// TIA Portal V20 export
// export: Created 2025-12-01T14:56:48.2327628Z, ExportSetting None, DisplayName Totally Integrated Automation Portal, DisplayVersion V20 Update 3, DisplayName TIA Portal Openness, DisplayVersion V20 Update 3, DisplayName TIA Portal Version Control Interface, DisplayVersion V20 Update 3, DisplayName STEP 7 Professional, DisplayVersion V20 Update 3, DisplayName STEP 7 Safety, DisplayVersion V20 Update 2, DisplayName WinCC Basic/Comfort/Advanced, DisplayVersion V20 Update 3, DisplayName WinCC Professional, DisplayVersion V20 Update 3, DisplayName WinCC Unified, DisplayVersion V20 Update 3
FUNCTION_BLOCK "FB364_Mesa_ApiladorBandejas_ULMA"   // FB364, LAD
TITLE = Control del Ramal de Salidas
{ S7_Optimized_Access := 'FALSE' }
AUTHOR : TE_FSS
NAME : 20160211
VERSION : 3.2
// stored: AutoNumber false, SetENOAutomatically false
   VAR_INPUT
      Mesa : UInt;   // Mesa de la FB
      Error_Tx : Bool;   // Error en el Tx
      pHsMx : Bool;   // pHs de la Mesa
      Avance_Tx : Bool;   // Avance de Tx
      TP_Up : Bool;   // Detector de TP Arriba
      TP_Down : Bool;   // Detector de TP Abajo
      PRV_AVTF_Bandeja : Bool;   // E1 >> Aviso de Entrada de Bandeja
      PRV_AVTF_Pila_Bandejas : Bool;   // E1 >> Aviso de Entrada de Pila
      NXT_Carga_OK : Bool;   // S3 >> Permiso de Salida
      DejarCargaEnMesa : Bool;   // Dejar la Bandeja En la Mesa
      V_pHsMx : Int;   // Valor de Presencia
      V_ApHsMx : Int;   // Valor de Ausencia
      V_TOut_Atasco : Int;   // Valor de TimeOut de Entrada
      V_TOut_TP : Int;   // Valor de TmeOut de Tope
      V_Vaciado : Int;   // Valor de Vaciado
   END_VAR
   VAR_OUTPUT
      PRV_Carga_OK : Bool;   // E1 >> Permiso de Entrada
      NXT_AVTF_Bandeja : Bool;   // S3 >> Aviso de Salida de Bandeja
      NXT_AVTF_Pila : Bool;   // S3 >> Aviso de Salida de Pila
   END_VAR
   VAR_IN_OUT
      Ord_ApilarBandeja : Bool;   // Orden de Apilar Bandeja
      Ord_SalidaPila : Bool;   // Orden de Salida de Pila
   END_VAR
   VAR
      Mx_ET00 : Bool;
      Mx_ET01 : Bool;
      Mx_ET02 : Bool;
      Mx_ET10 : Bool;
      Mx_ET11 : Bool;
      Mx_ET50 : Bool;   // Descarga de Bandeja
      Mx_ET51 : Bool;   // Descarga de Bandeja
      Mx_ET60 : Bool;   // Ciclo Apilado
      Mx_ET61 : Bool;   // Ciclo Apilado
      Mx_ET70 : Bool;   // Descarga De Pila de Bandejas
      Mx_ET71 : Bool;   // Descarga De Pila de Bandejas
      STAT_NXT_AVTF_Bandeja : Bool;   // Interna >> Aviso de Salida de Bandeja
      STAT_NXT_AVTF_Pila : Bool;   // Interna >> Aviso de Salida de Pila
      MA_Avanzar_Tx : Bool;
      MA_Parar_Tx : Bool;
      MA_Subir_TP : Bool;
      MA_Bajar_TP : Bool;
      CNT_pHsMx { S7_SetPoint := 'True'} : "FB910_CNT_UHS";
      CNT_ApHsMx { S7_SetPoint := 'True'} : "FB910_CNT_UHS";
      TMP_Vaciado { S7_SetPoint := 'True'} : "FB910_CNT_UHS";
      TOut_Atasco { S7_SetPoint := 'True'} : "FB910_CNT_UHS";
      TOut_Subir_TP { S7_SetPoint := 'True'} : "FB910_CNT_UHS";
      TOut_Bajar_TP { S7_SetPoint := 'True'} : "FB910_CNT_UHS";
   END_VAR
   VAR_TEMP
      EstadoZona : "EstadoZona";   // Estado de Zona de la Mesa
      EstadoVI : "EstadosMesa";   // Estado del Vehiculo Inteliguente de la Mesa
      ConfigFB : "UDT_ConfigFB";   // Configuracion de la FB de la Mesa
      Aux_ET00 : Bool;
   END_VAR
BEGIN

REGION Network 1: INICIALIZAR - Recoger las Variables de Estado de la Mesa
   // Se recoge - Estado_CBx
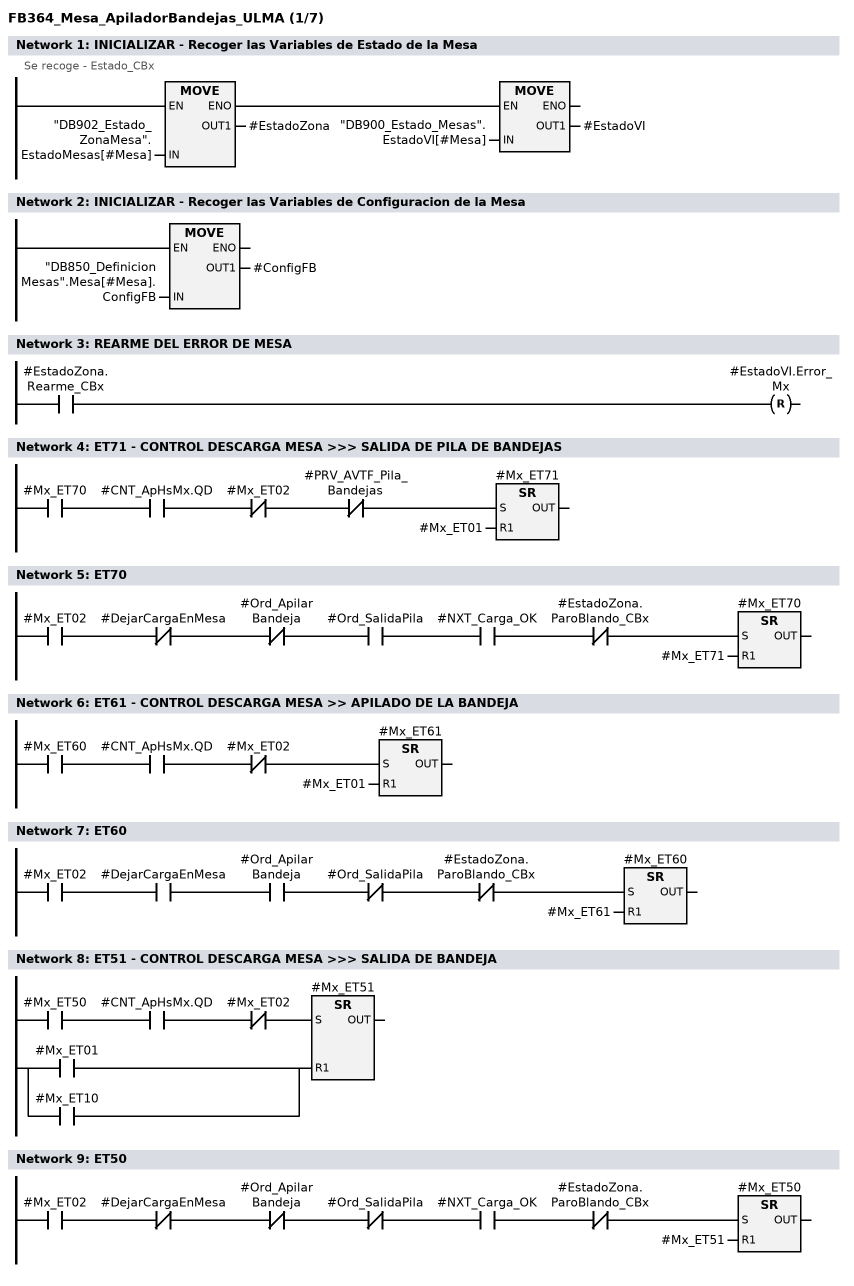
   RUNG wire#powerrail
      Move(in := "DB902_Estado_ZonaMesa".EstadoMesas[#Mesa], out1 => #EstadoZona)
      Move(in := "DB900_Estado_Mesas".EstadoVI[#Mesa], out1 => #EstadoVI)
   END_RUNG
   // the same network as SCL:
   #EstadoZona := "DB902_Estado_ZonaMesa".EstadoMesas[#Mesa];
   #EstadoVI := "DB900_Estado_Mesas".EstadoVI[#Mesa];
END_REGION

REGION Network 2: INICIALIZAR - Recoger las Variables de Configuracion de la Mesa
   RUNG wire#powerrail
      Move(in := "DB850_DefinicionMesas".Mesa[#Mesa].ConfigFB, out1 => #ConfigFB)
   END_RUNG
   // the same network as SCL:
   #ConfigFB := "DB850_DefinicionMesas".Mesa[#Mesa].ConfigFB;
END_REGION

REGION Network 3: REARME DEL ERROR DE MESA
   RUNG wire#powerrail
      Contact( #EstadoZona.Rearme_CBx )
      R_Coil( #EstadoVI.Error_Mx )
   END_RUNG
   // the same network as SCL:
   IF #EstadoZona.Rearme_CBx THEN #EstadoVI.Error_Mx := FALSE; END_IF;
END_REGION

REGION Network 4: ET71 - CONTROL DESCARGA MESA >>> SALIDA DE PILA DE BANDEJAS
   RUNG wire#powerrail
      Contact( #Mx_ET70 )
      Contact( #CNT_ApHsMx.QD )
      I_Contact( #Mx_ET02 )
      I_Contact( #PRV_AVTF_Pila_Bandejas )
      S_SR(operand := #Mx_ET71, r1 := #Mx_ET01)
   END_RUNG
   // the same network as SCL:
   IF #Mx_ET70 AND #CNT_ApHsMx.QD AND NOT #Mx_ET02 AND NOT #PRV_AVTF_Pila_Bandejas THEN
       #Mx_ET71 := TRUE;   // SR flip-flop
   END_IF;
   IF #Mx_ET01 THEN #Mx_ET71 := FALSE; END_IF;
END_REGION

REGION Network 5: ET70
   RUNG wire#powerrail
      Contact( #Mx_ET02 )
      I_Contact( #DejarCargaEnMesa )
      I_Contact( #Ord_ApilarBandeja )
      Contact( #Ord_SalidaPila )
      Contact( #NXT_Carga_OK )
      I_Contact( #EstadoZona.ParoBlando_CBx )
      S_SR(operand := #Mx_ET70, r1 := #Mx_ET71)
   END_RUNG
   // the same network as SCL:
   IF #Mx_ET02 AND NOT #DejarCargaEnMesa AND NOT #Ord_ApilarBandeja AND #Ord_SalidaPila AND #NXT_Carga_OK AND NOT #EstadoZona.ParoBlando_CBx THEN
       #Mx_ET70 := TRUE;   // SR flip-flop
   END_IF;
   IF #Mx_ET71 THEN #Mx_ET70 := FALSE; END_IF;
END_REGION

REGION Network 6: ET61 - CONTROL DESCARGA MESA >> APILADO DE LA BANDEJA
   RUNG wire#powerrail
      Contact( #Mx_ET60 )
      Contact( #CNT_ApHsMx.QD )
      I_Contact( #Mx_ET02 )
      S_SR(operand := #Mx_ET61, r1 := #Mx_ET01)
   END_RUNG
   // the same network as SCL:
   IF #Mx_ET60 AND #CNT_ApHsMx.QD AND NOT #Mx_ET02 THEN
       #Mx_ET61 := TRUE;   // SR flip-flop
   END_IF;
   IF #Mx_ET01 THEN #Mx_ET61 := FALSE; END_IF;
END_REGION

REGION Network 7: ET60
   RUNG wire#powerrail
      Contact( #Mx_ET02 )
      Contact( #DejarCargaEnMesa )
      Contact( #Ord_ApilarBandeja )
      I_Contact( #Ord_SalidaPila )
      I_Contact( #EstadoZona.ParoBlando_CBx )
      S_SR(operand := #Mx_ET60, r1 := #Mx_ET61)
   END_RUNG
   // the same network as SCL:
   IF #Mx_ET02 AND #DejarCargaEnMesa AND #Ord_ApilarBandeja AND NOT #Ord_SalidaPila AND NOT #EstadoZona.ParoBlando_CBx THEN
       #Mx_ET60 := TRUE;   // SR flip-flop
   END_IF;
   IF #Mx_ET61 THEN #Mx_ET60 := FALSE; END_IF;
END_REGION

REGION Network 8: ET51 - CONTROL DESCARGA MESA >>> SALIDA DE BANDEJA
   RUNG wire#powerrail
      Contact( #Mx_ET50 )
      Contact( #CNT_ApHsMx.QD )
      I_Contact( #Mx_ET02 )
      S_SR(operand := #Mx_ET51, r1 := wire#w1)
   END_RUNG
   RUNG wire#powerrail
      Contact( #Mx_ET01 )
   END_RUNG wire#w1
   RUNG wire#powerrail
      Contact( #Mx_ET10 )
   END_RUNG wire#w1
   // the same network as SCL:
   IF #Mx_ET50 AND #CNT_ApHsMx.QD AND NOT #Mx_ET02 THEN
       #Mx_ET51 := TRUE;   // SR flip-flop
   END_IF;
   IF #Mx_ET01 OR #Mx_ET10 THEN #Mx_ET51 := FALSE; END_IF;
END_REGION

REGION Network 9: ET50
   RUNG wire#powerrail
      Contact( #Mx_ET02 )
      I_Contact( #DejarCargaEnMesa )
      I_Contact( #Ord_ApilarBandeja )
      I_Contact( #Ord_SalidaPila )
      Contact( #NXT_Carga_OK )
      I_Contact( #EstadoZona.ParoBlando_CBx )
      S_SR(operand := #Mx_ET50, r1 := #Mx_ET51)
   END_RUNG
   // the same network as SCL:
   IF #Mx_ET02 AND NOT #DejarCargaEnMesa AND NOT #Ord_ApilarBandeja AND NOT #Ord_SalidaPila AND #NXT_Carga_OK AND NOT #EstadoZona.ParoBlando_CBx THEN
       #Mx_ET50 := TRUE;   // SR flip-flop
   END_IF;
   IF #Mx_ET51 THEN #Mx_ET50 := FALSE; END_IF;
END_REGION

REGION Network 10: ET02 - ESTADO REPOSO CARGADA
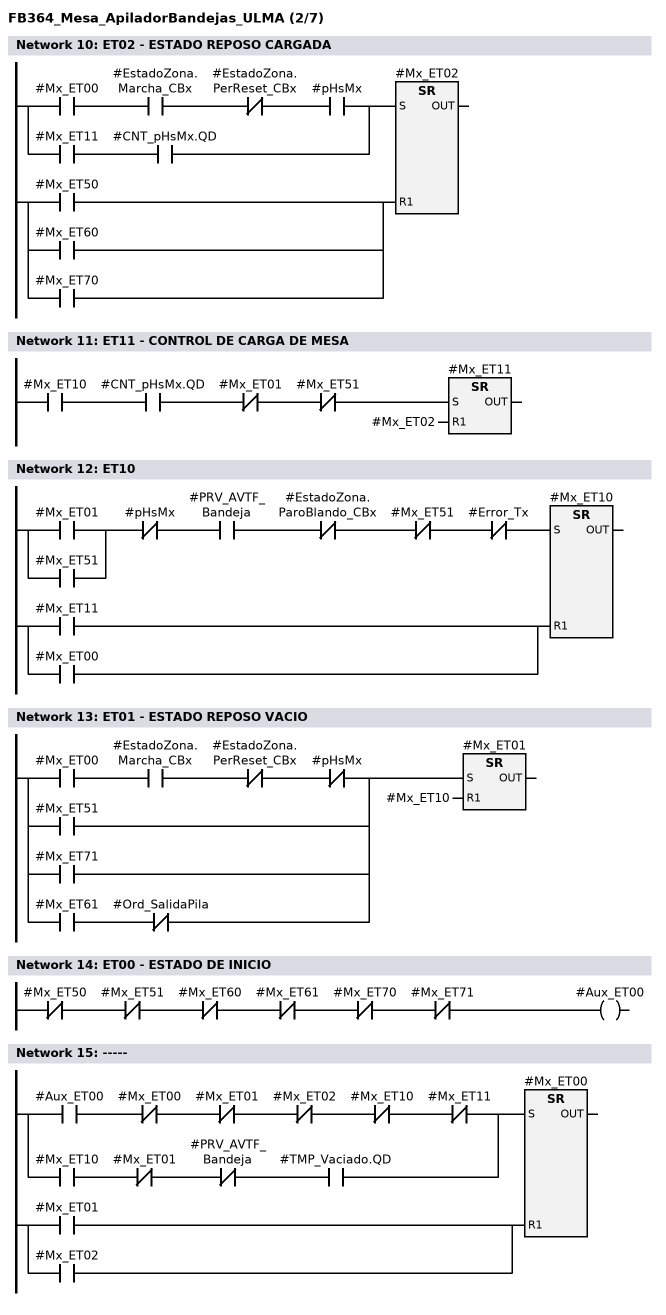
   RUNG wire#powerrail
      Contact( #Mx_ET00 )
      Contact( #EstadoZona.Marcha_CBx )
      I_Contact( #EstadoZona.PerReset_CBx )
      Contact( #pHsMx )
      wire#w1
      S_SR(operand := #Mx_ET02, r1 := wire#w2)
   END_RUNG
   RUNG wire#powerrail
      Contact( #Mx_ET11 )
      Contact( #CNT_pHsMx.QD )
   END_RUNG wire#w1
   RUNG wire#powerrail
      Contact( #Mx_ET50 )
   END_RUNG wire#w2
   RUNG wire#powerrail
      Contact( #Mx_ET60 )
   END_RUNG wire#w2
   RUNG wire#powerrail
      Contact( #Mx_ET70 )
   END_RUNG wire#w2
   // the same network as SCL:
   IF (#Mx_ET00 AND #EstadoZona.Marcha_CBx AND NOT #EstadoZona.PerReset_CBx AND #pHsMx) OR (#Mx_ET11 AND #CNT_pHsMx.QD) THEN
       #Mx_ET02 := TRUE;   // SR flip-flop
   END_IF;
   IF #Mx_ET50 OR #Mx_ET60 OR #Mx_ET70 THEN #Mx_ET02 := FALSE; END_IF;
END_REGION

REGION Network 11: ET11 - CONTROL DE CARGA DE MESA
   RUNG wire#powerrail
      Contact( #Mx_ET10 )
      Contact( #CNT_pHsMx.QD )
      I_Contact( #Mx_ET01 )
      I_Contact( #Mx_ET51 )
      S_SR(operand := #Mx_ET11, r1 := #Mx_ET02)
   END_RUNG
   // the same network as SCL:
   IF #Mx_ET10 AND #CNT_pHsMx.QD AND NOT #Mx_ET01 AND NOT #Mx_ET51 THEN
       #Mx_ET11 := TRUE;   // SR flip-flop
   END_IF;
   IF #Mx_ET02 THEN #Mx_ET11 := FALSE; END_IF;
END_REGION

REGION Network 12: ET10
   RUNG wire#powerrail
      Contact( #Mx_ET01 )
      wire#w1
      I_Contact( #pHsMx )
      Contact( #PRV_AVTF_Bandeja )
      I_Contact( #EstadoZona.ParoBlando_CBx )
      I_Contact( #Mx_ET51 )
      I_Contact( #Error_Tx )
      S_SR(operand := #Mx_ET10, r1 := wire#w2)
   END_RUNG
   RUNG wire#powerrail
      Contact( #Mx_ET51 )
   END_RUNG wire#w1
   RUNG wire#powerrail
      Contact( #Mx_ET11 )
   END_RUNG wire#w2
   RUNG wire#powerrail
      Contact( #Mx_ET00 )
   END_RUNG wire#w2
   // the same network as SCL:
   IF (#Mx_ET01 OR #Mx_ET51) AND NOT #pHsMx AND #PRV_AVTF_Bandeja AND NOT #EstadoZona.ParoBlando_CBx AND NOT #Mx_ET51 AND NOT #Error_Tx THEN
       #Mx_ET10 := TRUE;   // SR flip-flop
   END_IF;
   IF #Mx_ET11 OR #Mx_ET00 THEN #Mx_ET10 := FALSE; END_IF;
END_REGION

REGION Network 13: ET01 - ESTADO REPOSO VACIO
   RUNG wire#powerrail
      Contact( #Mx_ET00 )
      Contact( #EstadoZona.Marcha_CBx )
      I_Contact( #EstadoZona.PerReset_CBx )
      I_Contact( #pHsMx )
      wire#w1
      S_SR(operand := #Mx_ET01, r1 := #Mx_ET10)
   END_RUNG
   RUNG wire#powerrail
      Contact( #Mx_ET51 )
   END_RUNG wire#w1
   RUNG wire#powerrail
      Contact( #Mx_ET71 )
   END_RUNG wire#w1
   RUNG wire#powerrail
      Contact( #Mx_ET61 )
      I_Contact( #Ord_SalidaPila )
   END_RUNG wire#w1
   // the same network as SCL:
   IF (#Mx_ET00 AND #EstadoZona.Marcha_CBx AND NOT #EstadoZona.PerReset_CBx AND NOT #pHsMx) OR #Mx_ET51 OR #Mx_ET71 OR (#Mx_ET61 AND NOT #Ord_SalidaPila) THEN
       #Mx_ET01 := TRUE;   // SR flip-flop
   END_IF;
   IF #Mx_ET10 THEN #Mx_ET01 := FALSE; END_IF;
END_REGION

REGION Network 14: ET00 - ESTADO DE INICIO
   RUNG wire#powerrail
      I_Contact( #Mx_ET50 )
      I_Contact( #Mx_ET51 )
      I_Contact( #Mx_ET60 )
      I_Contact( #Mx_ET61 )
      I_Contact( #Mx_ET70 )
      I_Contact( #Mx_ET71 )
      Coil( #Aux_ET00 )
   END_RUNG
   // the same network as SCL:
   #Aux_ET00 := NOT #Mx_ET50 AND NOT #Mx_ET51 AND NOT #Mx_ET60 AND NOT #Mx_ET61 AND NOT #Mx_ET70 AND NOT #Mx_ET71;
END_REGION

REGION Network 15: -----
   RUNG wire#powerrail
      Contact( #Aux_ET00 )
      I_Contact( #Mx_ET00 )
      I_Contact( #Mx_ET01 )
      I_Contact( #Mx_ET02 )
      I_Contact( #Mx_ET10 )
      I_Contact( #Mx_ET11 )
      wire#w1
      S_SR(operand := #Mx_ET00, r1 := wire#w2)
   END_RUNG
   RUNG wire#powerrail
      Contact( #Mx_ET10 )
      I_Contact( #Mx_ET01 )
      I_Contact( #PRV_AVTF_Bandeja )
      Contact( #TMP_Vaciado.QD )
   END_RUNG wire#w1
   RUNG wire#powerrail
      Contact( #Mx_ET01 )
   END_RUNG wire#w2
   RUNG wire#powerrail
      Contact( #Mx_ET02 )
   END_RUNG wire#w2
   // the same network as SCL:
   IF (#Aux_ET00 AND NOT #Mx_ET00 AND NOT #Mx_ET01 AND NOT #Mx_ET02 AND NOT #Mx_ET10 AND NOT #Mx_ET11) OR (#Mx_ET10 AND NOT #Mx_ET01 AND NOT #PRV_AVTF_Bandeja AND #TMP_Vaciado.QD) THEN
       #Mx_ET00 := TRUE;   // SR flip-flop
   END_IF;
   IF #Mx_ET01 OR #Mx_ET02 THEN #Mx_ET00 := FALSE; END_IF;
END_REGION

REGION Network 16: CONTADOR DE PRESENCIA
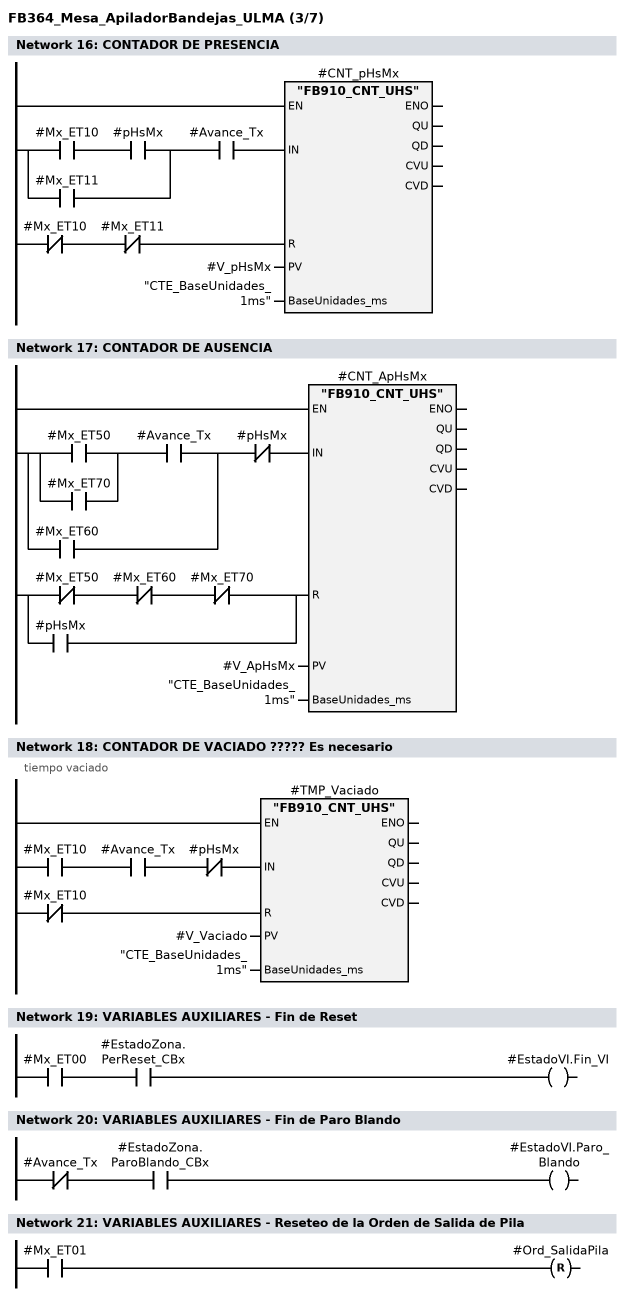
   RUNG wire#powerrail
      #CNT_pHsMx(IN := wire#w2, R := wire#w3, PV := #V_pHsMx, BaseUnidades_ms := "CTE_BaseUnidades_1ms", QU =>, QD =>, CVU =>, CVD =>)
   END_RUNG
   RUNG wire#powerrail
      Contact( #Mx_ET10 )
      Contact( #pHsMx )
      wire#w1
      Contact( #Avance_Tx )
   END_RUNG wire#w2
   RUNG wire#powerrail
      Contact( #Mx_ET11 )
   END_RUNG wire#w1
   RUNG wire#powerrail
      I_Contact( #Mx_ET10 )
      I_Contact( #Mx_ET11 )
   END_RUNG wire#w3
   // the same network as SCL:
   #CNT_pHsMx(IN := ((#Mx_ET10 AND #pHsMx) OR #Mx_ET11) AND #Avance_Tx,   // "FB910_CNT_UHS"
              R := NOT #Mx_ET10 AND NOT #Mx_ET11,
              PV := #V_pHsMx,
              BaseUnidades_ms := "CTE_BaseUnidades_1ms");
END_REGION

REGION Network 17: CONTADOR DE AUSENCIA
   RUNG wire#powerrail
      #CNT_ApHsMx(IN := wire#w3, R := wire#w4, PV := #V_ApHsMx, BaseUnidades_ms := "CTE_BaseUnidades_1ms", QU =>, QD =>, CVU =>, CVD =>)
   END_RUNG
   RUNG wire#powerrail
      Contact( #Mx_ET50 )
      wire#w1
      Contact( #Avance_Tx )
      wire#w2
      I_Contact( #pHsMx )
   END_RUNG wire#w3
   RUNG wire#powerrail
      Contact( #Mx_ET70 )
   END_RUNG wire#w1
   RUNG wire#powerrail
      Contact( #Mx_ET60 )
   END_RUNG wire#w2
   RUNG wire#powerrail
      I_Contact( #Mx_ET50 )
      I_Contact( #Mx_ET60 )
      I_Contact( #Mx_ET70 )
   END_RUNG wire#w4
   RUNG wire#powerrail
      Contact( #pHsMx )
   END_RUNG wire#w4
   // the same network as SCL:
   #CNT_ApHsMx(IN := (((#Mx_ET50 OR #Mx_ET70) AND #Avance_Tx) OR #Mx_ET60) AND NOT #pHsMx,   // "FB910_CNT_UHS"
               R := (NOT #Mx_ET50 AND NOT #Mx_ET60 AND NOT #Mx_ET70) OR #pHsMx,
               PV := #V_ApHsMx,
               BaseUnidades_ms := "CTE_BaseUnidades_1ms");
END_REGION

REGION Network 18: CONTADOR DE VACIADO ????? Es necesario
   // tiempo vaciado
   RUNG wire#powerrail
      #TMP_Vaciado(IN := wire#w1, R := wire#w2, PV := #V_Vaciado, BaseUnidades_ms := "CTE_BaseUnidades_1ms", QU =>, QD =>, CVU =>, CVD =>)
   END_RUNG
   RUNG wire#powerrail
      Contact( #Mx_ET10 )
      Contact( #Avance_Tx )
      I_Contact( #pHsMx )
   END_RUNG wire#w1
   RUNG wire#powerrail
      I_Contact( #Mx_ET10 )
   END_RUNG wire#w2
   // the same network as SCL:
   #TMP_Vaciado(IN := #Mx_ET10 AND #Avance_Tx AND NOT #pHsMx,   // "FB910_CNT_UHS"
                R := NOT #Mx_ET10,
                PV := #V_Vaciado,
                BaseUnidades_ms := "CTE_BaseUnidades_1ms");
END_REGION

REGION Network 19: VARIABLES AUXILIARES - Fin de Reset
   RUNG wire#powerrail
      Contact( #Mx_ET00 )
      Contact( #EstadoZona.PerReset_CBx )
      Coil( #EstadoVI.Fin_VI )
   END_RUNG
   // the same network as SCL:
   #EstadoVI.Fin_VI := #Mx_ET00 AND #EstadoZona.PerReset_CBx;
END_REGION

REGION Network 20: VARIABLES AUXILIARES - Fin de Paro Blando
   RUNG wire#powerrail
      I_Contact( #Avance_Tx )
      Contact( #EstadoZona.ParoBlando_CBx )
      Coil( #EstadoVI.Paro_Blando )
   END_RUNG
   // the same network as SCL:
   #EstadoVI.Paro_Blando := NOT #Avance_Tx AND #EstadoZona.ParoBlando_CBx;
END_REGION

REGION Network 21: VARIABLES AUXILIARES - Reseteo de la Orden de Salida de Pila
   RUNG wire#powerrail
      Contact( #Mx_ET01 )
      R_Coil( #Ord_SalidaPila )
   END_RUNG
   // the same network as SCL:
   IF #Mx_ET01 THEN #Ord_SalidaPila := FALSE; END_IF;
END_REGION

REGION Network 22: VARIABLES AUXILIARES - Permiso de Entrada - PRV_Carga_OK
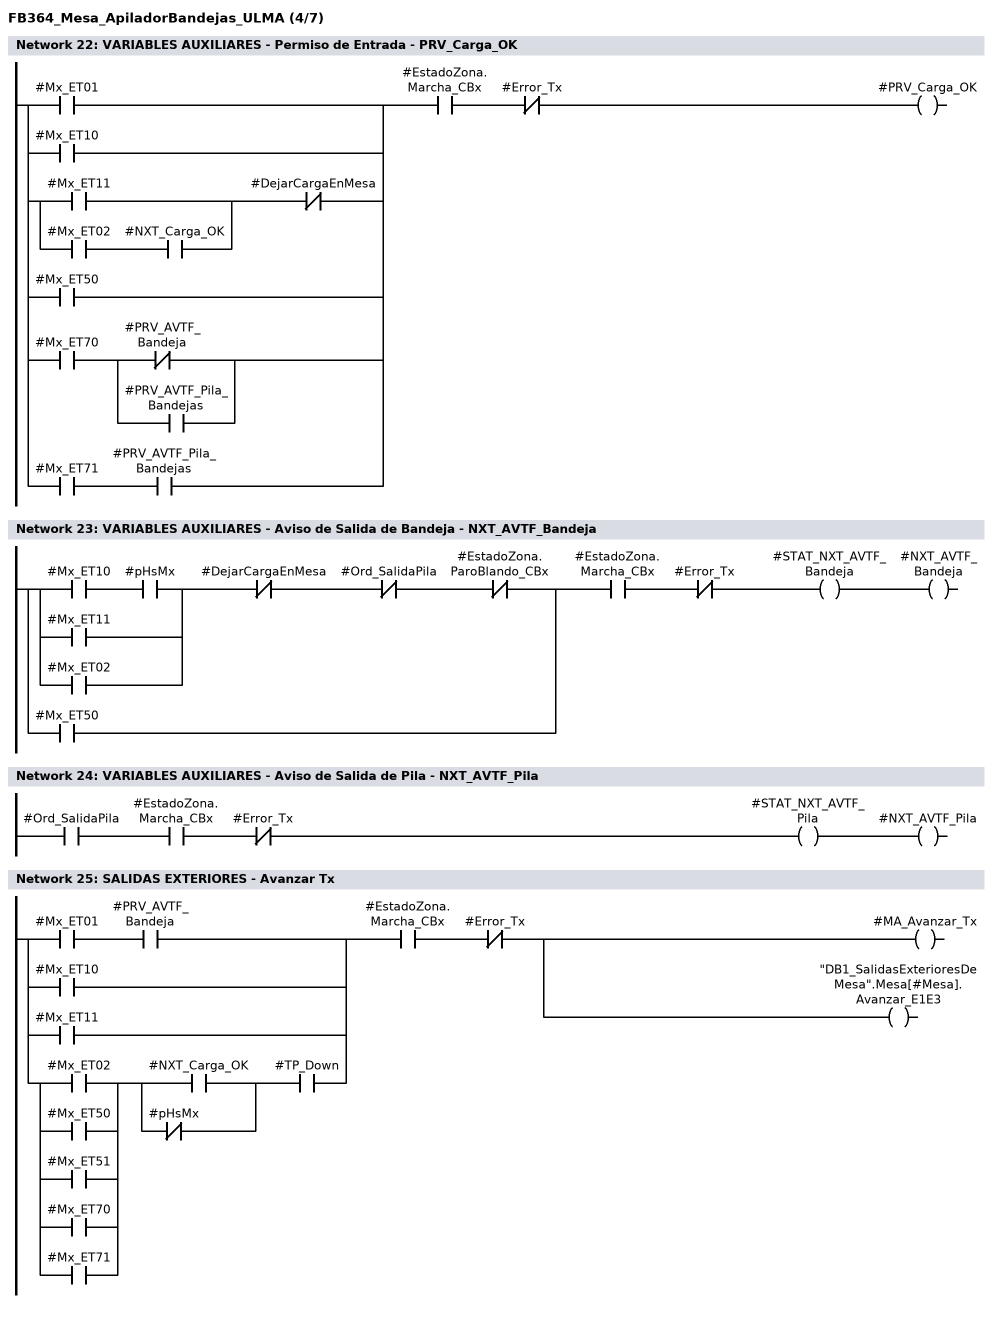
   RUNG wire#powerrail
      Contact( #Mx_ET01 )
      wire#w1
      Contact( #EstadoZona.Marcha_CBx )
      I_Contact( #Error_Tx )
      Coil( #PRV_Carga_OK )
   END_RUNG
   RUNG wire#powerrail
      Contact( #Mx_ET10 )
   END_RUNG wire#w1
   RUNG wire#powerrail
      Contact( #Mx_ET11 )
      wire#w2
      I_Contact( #DejarCargaEnMesa )
   END_RUNG wire#w1
   RUNG wire#powerrail
      Contact( #Mx_ET02 )
      Contact( #NXT_Carga_OK )
   END_RUNG wire#w2
   RUNG wire#powerrail
      Contact( #Mx_ET50 )
   END_RUNG wire#w1
   RUNG wire#powerrail
      Contact( #Mx_ET70 )
      wire#w3
      I_Contact( #PRV_AVTF_Bandeja )
   END_RUNG wire#w1
   RUNG wire#w3
      Contact( #PRV_AVTF_Pila_Bandejas )
   END_RUNG wire#w1
   RUNG wire#powerrail
      Contact( #Mx_ET71 )
      Contact( #PRV_AVTF_Pila_Bandejas )
   END_RUNG wire#w1
   // the same network as SCL:
   #PRV_Carga_OK := (#Mx_ET01 OR #Mx_ET10 OR ((#Mx_ET11 OR (#Mx_ET02 AND #NXT_Carga_OK)) AND NOT #DejarCargaEnMesa) OR #Mx_ET50 OR (#Mx_ET70 AND (NOT #PRV_AVTF_Bandeja OR #PRV_AVTF_Pila_Bandejas)) OR (#Mx_ET71 AND #PRV_AVTF_Pila_Bandejas)) AND #EstadoZona.Marcha_CBx AND NOT #Error_Tx;
END_REGION

REGION Network 23: VARIABLES AUXILIARES - Aviso de Salida de Bandeja - NXT_AVTF_Bandeja
   RUNG wire#powerrail
      Contact( #Mx_ET10 )
      Contact( #pHsMx )
      wire#w1
      I_Contact( #DejarCargaEnMesa )
      I_Contact( #Ord_SalidaPila )
      I_Contact( #EstadoZona.ParoBlando_CBx )
      wire#w2
      Contact( #EstadoZona.Marcha_CBx )
      I_Contact( #Error_Tx )
      Coil( #STAT_NXT_AVTF_Bandeja )
      Coil( #NXT_AVTF_Bandeja )
   END_RUNG
   RUNG wire#powerrail
      Contact( #Mx_ET11 )
   END_RUNG wire#w1
   RUNG wire#powerrail
      Contact( #Mx_ET02 )
   END_RUNG wire#w1
   RUNG wire#powerrail
      Contact( #Mx_ET50 )
   END_RUNG wire#w2
   // the same network as SCL:
   #STAT_NXT_AVTF_Bandeja := ((((#Mx_ET10 AND #pHsMx) OR #Mx_ET11 OR #Mx_ET02) AND NOT #DejarCargaEnMesa AND NOT #Ord_SalidaPila AND NOT #EstadoZona.ParoBlando_CBx) OR #Mx_ET50) AND #EstadoZona.Marcha_CBx AND NOT #Error_Tx;
   #NXT_AVTF_Bandeja := #STAT_NXT_AVTF_Bandeja;
END_REGION

REGION Network 24: VARIABLES AUXILIARES - Aviso de Salida de Pila - NXT_AVTF_Pila
   RUNG wire#powerrail
      Contact( #Ord_SalidaPila )
      Contact( #EstadoZona.Marcha_CBx )
      I_Contact( #Error_Tx )
      Coil( #STAT_NXT_AVTF_Pila )
      Coil( #NXT_AVTF_Pila )
   END_RUNG
   // the same network as SCL:
   #STAT_NXT_AVTF_Pila := #Ord_SalidaPila AND #EstadoZona.Marcha_CBx AND NOT #Error_Tx;
   #NXT_AVTF_Pila := #STAT_NXT_AVTF_Pila;
END_REGION

REGION Network 25: SALIDAS EXTERIORES - Avanzar Tx
   RUNG wire#powerrail
      Contact( #Mx_ET01 )
      Contact( #PRV_AVTF_Bandeja )
      wire#w1
      Contact( #EstadoZona.Marcha_CBx )
      I_Contact( #Error_Tx )
      wire#w4
      Coil( #MA_Avanzar_Tx )
   END_RUNG
   RUNG wire#powerrail
      Contact( #Mx_ET10 )
   END_RUNG wire#w1
   RUNG wire#powerrail
      Contact( #Mx_ET11 )
   END_RUNG wire#w1
   RUNG wire#powerrail
      Contact( #Mx_ET02 )
      wire#w2
      Contact( #NXT_Carga_OK )
      wire#w3
      Contact( #TP_Down )
   END_RUNG wire#w1
   RUNG wire#powerrail
      Contact( #Mx_ET50 )
   END_RUNG wire#w2
   RUNG wire#powerrail
      Contact( #Mx_ET51 )
   END_RUNG wire#w2
   RUNG wire#powerrail
      Contact( #Mx_ET70 )
   END_RUNG wire#w2
   RUNG wire#powerrail
      Contact( #Mx_ET71 )
   END_RUNG wire#w2
   RUNG wire#w2
      I_Contact( #pHsMx )
   END_RUNG wire#w3
   RUNG wire#w4
      Coil( "DB1_SalidasExterioresDeMesa".Mesa[#Mesa].Avanzar_E1E3 )
   END_RUNG
   // the same network as SCL:
   #MA_Avanzar_Tx := ((#Mx_ET01 AND #PRV_AVTF_Bandeja) OR #Mx_ET10 OR #Mx_ET11 OR ((#Mx_ET02 OR #Mx_ET50 OR #Mx_ET51 OR #Mx_ET70 OR #Mx_ET71) AND (#NXT_Carga_OK OR NOT #pHsMx) AND #TP_Down)) AND #EstadoZona.Marcha_CBx AND NOT #Error_Tx;
   "DB1_SalidasExterioresDeMesa".Mesa[#Mesa].Avanzar_E1E3 := #MA_Avanzar_Tx;
END_REGION

REGION Network 26: SALIDAS EXTERIORES - Parar Tx
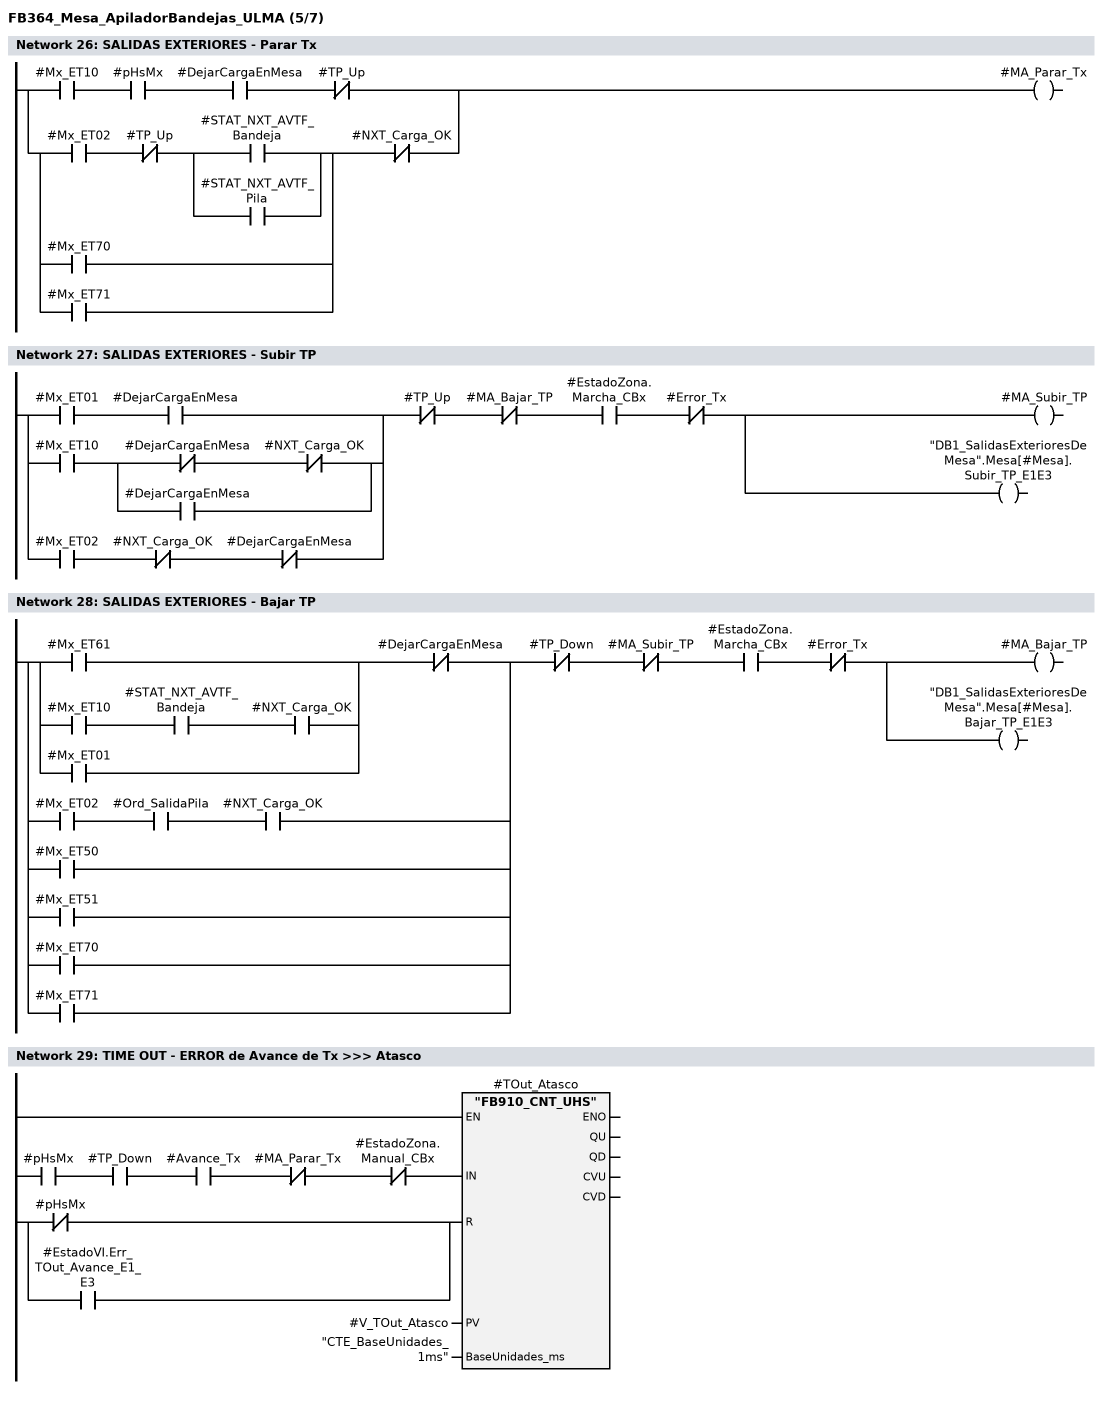
   RUNG wire#powerrail
      Contact( #Mx_ET10 )
      Contact( #pHsMx )
      Contact( #DejarCargaEnMesa )
      I_Contact( #TP_Up )
      wire#w1
      Coil( #MA_Parar_Tx )
   END_RUNG
   RUNG wire#powerrail
      Contact( #Mx_ET02 )
      I_Contact( #TP_Up )
      wire#w2
      Contact( #STAT_NXT_AVTF_Bandeja )
      wire#w3
      I_Contact( #NXT_Carga_OK )
   END_RUNG wire#w1
   RUNG wire#w2
      Contact( #STAT_NXT_AVTF_Pila )
   END_RUNG wire#w3
   RUNG wire#powerrail
      Contact( #Mx_ET70 )
   END_RUNG wire#w3
   RUNG wire#powerrail
      Contact( #Mx_ET71 )
   END_RUNG wire#w3
   // the same network as SCL:
   #MA_Parar_Tx := (#Mx_ET10 AND #pHsMx AND #DejarCargaEnMesa AND NOT #TP_Up) OR (((#Mx_ET02 AND NOT #TP_Up AND (#STAT_NXT_AVTF_Bandeja OR #STAT_NXT_AVTF_Pila)) OR #Mx_ET70 OR #Mx_ET71) AND NOT #NXT_Carga_OK);
END_REGION

REGION Network 27: SALIDAS EXTERIORES - Subir TP
   RUNG wire#powerrail
      Contact( #Mx_ET01 )
      Contact( #DejarCargaEnMesa )
      wire#w1
      I_Contact( #TP_Up )
      I_Contact( #MA_Bajar_TP )
      Contact( #EstadoZona.Marcha_CBx )
      I_Contact( #Error_Tx )
      wire#w3
      Coil( #MA_Subir_TP )
   END_RUNG
   RUNG wire#powerrail
      Contact( #Mx_ET10 )
      wire#w2
      I_Contact( #DejarCargaEnMesa )
      I_Contact( #NXT_Carga_OK )
   END_RUNG wire#w1
   RUNG wire#w2
      Contact( #DejarCargaEnMesa )
   END_RUNG wire#w1
   RUNG wire#powerrail
      Contact( #Mx_ET02 )
      I_Contact( #NXT_Carga_OK )
      I_Contact( #DejarCargaEnMesa )
   END_RUNG wire#w1
   RUNG wire#w3
      Coil( "DB1_SalidasExterioresDeMesa".Mesa[#Mesa].Subir_TP_E1E3 )
   END_RUNG
   // the same network as SCL:
   #MA_Subir_TP := ((#Mx_ET01 AND #DejarCargaEnMesa) OR (#Mx_ET10 AND ((NOT #DejarCargaEnMesa AND NOT #NXT_Carga_OK) OR #DejarCargaEnMesa)) OR (#Mx_ET02 AND NOT #NXT_Carga_OK AND NOT #DejarCargaEnMesa)) AND NOT #TP_Up AND NOT #MA_Bajar_TP AND #EstadoZona.Marcha_CBx AND NOT #Error_Tx;
   "DB1_SalidasExterioresDeMesa".Mesa[#Mesa].Subir_TP_E1E3 := #MA_Subir_TP;
END_REGION

REGION Network 28: SALIDAS EXTERIORES - Bajar TP
   RUNG wire#powerrail
      Contact( #Mx_ET61 )
      wire#w1
      I_Contact( #DejarCargaEnMesa )
      wire#w2
      I_Contact( #TP_Down )
      I_Contact( #MA_Subir_TP )
      Contact( #EstadoZona.Marcha_CBx )
      I_Contact( #Error_Tx )
      wire#w3
      Coil( #MA_Bajar_TP )
   END_RUNG
   RUNG wire#powerrail
      Contact( #Mx_ET10 )
      Contact( #STAT_NXT_AVTF_Bandeja )
      Contact( #NXT_Carga_OK )
   END_RUNG wire#w1
   RUNG wire#powerrail
      Contact( #Mx_ET01 )
   END_RUNG wire#w1
   RUNG wire#powerrail
      Contact( #Mx_ET02 )
      Contact( #Ord_SalidaPila )
      Contact( #NXT_Carga_OK )
   END_RUNG wire#w2
   RUNG wire#powerrail
      Contact( #Mx_ET50 )
   END_RUNG wire#w2
   RUNG wire#powerrail
      Contact( #Mx_ET51 )
   END_RUNG wire#w2
   RUNG wire#powerrail
      Contact( #Mx_ET70 )
   END_RUNG wire#w2
   RUNG wire#powerrail
      Contact( #Mx_ET71 )
   END_RUNG wire#w2
   RUNG wire#w3
      Coil( "DB1_SalidasExterioresDeMesa".Mesa[#Mesa].Bajar_TP_E1E3 )
   END_RUNG
   // the same network as SCL:
   #MA_Bajar_TP := (((#Mx_ET61 OR (#Mx_ET10 AND #STAT_NXT_AVTF_Bandeja AND #NXT_Carga_OK) OR #Mx_ET01) AND NOT #DejarCargaEnMesa) OR (#Mx_ET02 AND #Ord_SalidaPila AND #NXT_Carga_OK) OR #Mx_ET50 OR #Mx_ET51 OR #Mx_ET70 OR #Mx_ET71) AND NOT #TP_Down AND NOT #MA_Subir_TP AND #EstadoZona.Marcha_CBx AND NOT #Error_Tx;
   "DB1_SalidasExterioresDeMesa".Mesa[#Mesa].Bajar_TP_E1E3 := #MA_Bajar_TP;
END_REGION

REGION Network 29: TIME OUT - ERROR de Avance de Tx >>> Atasco
   RUNG wire#powerrail
      #TOut_Atasco(IN := wire#w1, R := wire#w2, PV := #V_TOut_Atasco, BaseUnidades_ms := "CTE_BaseUnidades_1ms", QU =>, QD =>, CVU =>, CVD =>)
   END_RUNG
   RUNG wire#powerrail
      Contact( #pHsMx )
      Contact( #TP_Down )
      Contact( #Avance_Tx )
      I_Contact( #MA_Parar_Tx )
      I_Contact( #EstadoZona.Manual_CBx )
   END_RUNG wire#w1
   RUNG wire#powerrail
      I_Contact( #pHsMx )
   END_RUNG wire#w2
   RUNG wire#powerrail
      Contact( #EstadoVI.Err_TOut_Avance_E1_E3 )
   END_RUNG wire#w2
   // the same network as SCL:
   #TOut_Atasco(IN := #pHsMx AND #TP_Down AND #Avance_Tx AND NOT #MA_Parar_Tx AND NOT #EstadoZona.Manual_CBx,   // "FB910_CNT_UHS"
                R := NOT #pHsMx OR #EstadoVI.Err_TOut_Avance_E1_E3,
                PV := #V_TOut_Atasco,
                BaseUnidades_ms := "CTE_BaseUnidades_1ms");
END_REGION

REGION Network 30: ERROR de Avance de Tx >>> Atasco
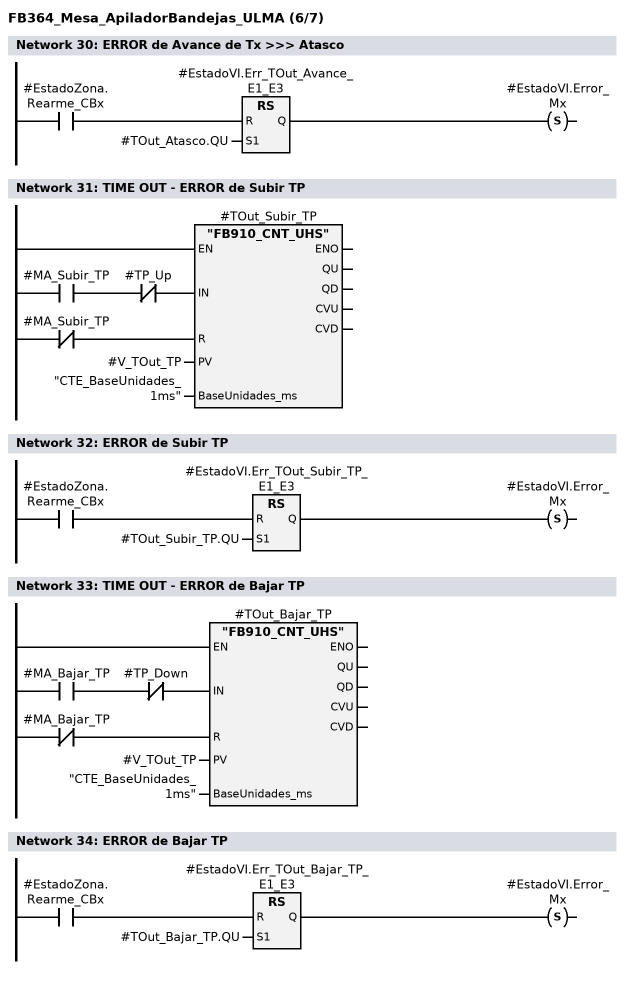
   RUNG wire#powerrail
      Contact( #EstadoZona.Rearme_CBx )
      S_RS(operand := #EstadoVI.Err_TOut_Avance_E1_E3, s1 := #TOut_Atasco.QU)
      S_Coil( #EstadoVI.Error_Mx )
   END_RUNG
   // the same network as SCL:
   IF #EstadoZona.Rearme_CBx THEN
       #EstadoVI.Err_TOut_Avance_E1_E3 := FALSE;   // RS flip-flop
   END_IF;
   IF #TOut_Atasco.QU THEN #EstadoVI.Err_TOut_Avance_E1_E3 := TRUE; END_IF;
   IF #EstadoVI.Err_TOut_Avance_E1_E3 THEN #EstadoVI.Error_Mx := TRUE; END_IF;
END_REGION

REGION Network 31: TIME OUT - ERROR de Subir TP
   RUNG wire#powerrail
      #TOut_Subir_TP(IN := wire#w1, R := wire#w2, PV := #V_TOut_TP, BaseUnidades_ms := "CTE_BaseUnidades_1ms", QU =>, QD =>, CVU =>, CVD =>)
   END_RUNG
   RUNG wire#powerrail
      Contact( #MA_Subir_TP )
      I_Contact( #TP_Up )
   END_RUNG wire#w1
   RUNG wire#powerrail
      I_Contact( #MA_Subir_TP )
   END_RUNG wire#w2
   // the same network as SCL:
   #TOut_Subir_TP(IN := #MA_Subir_TP AND NOT #TP_Up,   // "FB910_CNT_UHS"
                  R := NOT #MA_Subir_TP,
                  PV := #V_TOut_TP,
                  BaseUnidades_ms := "CTE_BaseUnidades_1ms");
END_REGION

REGION Network 32: ERROR de Subir TP
   RUNG wire#powerrail
      Contact( #EstadoZona.Rearme_CBx )
      S_RS(operand := #EstadoVI.Err_TOut_Subir_TP_E1_E3, s1 := #TOut_Subir_TP.QU)
      S_Coil( #EstadoVI.Error_Mx )
   END_RUNG
   // the same network as SCL:
   IF #EstadoZona.Rearme_CBx THEN
       #EstadoVI.Err_TOut_Subir_TP_E1_E3 := FALSE;   // RS flip-flop
   END_IF;
   IF #TOut_Subir_TP.QU THEN #EstadoVI.Err_TOut_Subir_TP_E1_E3 := TRUE; END_IF;
   IF #EstadoVI.Err_TOut_Subir_TP_E1_E3 THEN #EstadoVI.Error_Mx := TRUE; END_IF;
END_REGION

REGION Network 33: TIME OUT - ERROR de Bajar TP
   RUNG wire#powerrail
      #TOut_Bajar_TP(IN := wire#w1, R := wire#w2, PV := #V_TOut_TP, BaseUnidades_ms := "CTE_BaseUnidades_1ms", QU =>, QD =>, CVU =>, CVD =>)
   END_RUNG
   RUNG wire#powerrail
      Contact( #MA_Bajar_TP )
      I_Contact( #TP_Down )
   END_RUNG wire#w1
   RUNG wire#powerrail
      I_Contact( #MA_Bajar_TP )
   END_RUNG wire#w2
   // the same network as SCL:
   #TOut_Bajar_TP(IN := #MA_Bajar_TP AND NOT #TP_Down,   // "FB910_CNT_UHS"
                  R := NOT #MA_Bajar_TP,
                  PV := #V_TOut_TP,
                  BaseUnidades_ms := "CTE_BaseUnidades_1ms");
END_REGION

REGION Network 34: ERROR de Bajar TP
   RUNG wire#powerrail
      Contact( #EstadoZona.Rearme_CBx )
      S_RS(operand := #EstadoVI.Err_TOut_Bajar_TP_E1_E3, s1 := #TOut_Bajar_TP.QU)
      S_Coil( #EstadoVI.Error_Mx )
   END_RUNG
   // the same network as SCL:
   IF #EstadoZona.Rearme_CBx THEN
       #EstadoVI.Err_TOut_Bajar_TP_E1_E3 := FALSE;   // RS flip-flop
   END_IF;
   IF #TOut_Bajar_TP.QU THEN #EstadoVI.Err_TOut_Bajar_TP_E1_E3 := TRUE; END_IF;
   IF #EstadoVI.Err_TOut_Bajar_TP_E1_E3 THEN #EstadoVI.Error_Mx := TRUE; END_IF;
END_REGION

REGION Network 35: ESTADO DE LA MESA
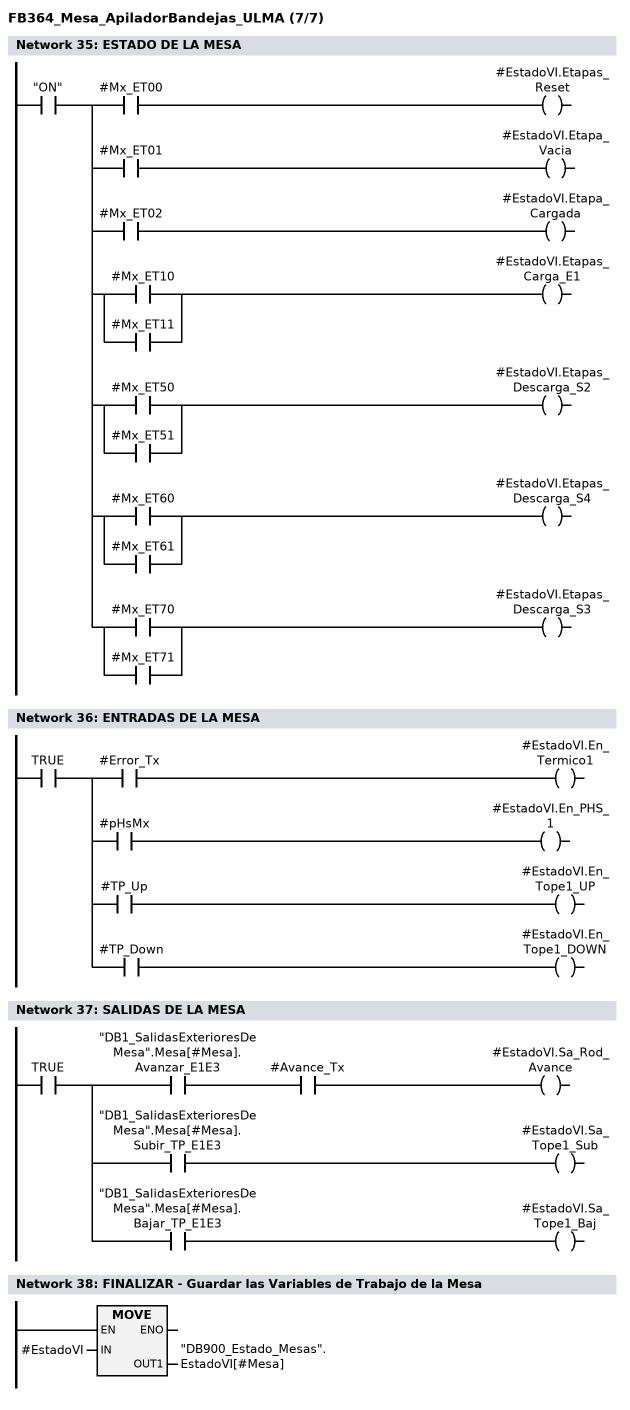
   RUNG wire#powerrail
      Contact( "ON" )
      wire#w1
      Contact( #Mx_ET00 )
      Coil( #EstadoVI.Etapas_Reset )
   END_RUNG
   RUNG wire#w1
      Contact( #Mx_ET01 )
      Coil( #EstadoVI.Etapa_Vacia )
   END_RUNG
   RUNG wire#w1
      Contact( #Mx_ET02 )
      Coil( #EstadoVI.Etapa_Cargada )
   END_RUNG
   RUNG wire#w1
      Contact( #Mx_ET10 )
      wire#w2
      Coil( #EstadoVI.Etapas_Carga_E1 )
   END_RUNG
   RUNG wire#w1
      Contact( #Mx_ET11 )
   END_RUNG wire#w2
   RUNG wire#w1
      Contact( #Mx_ET50 )
      wire#w3
      Coil( #EstadoVI.Etapas_Descarga_S2 )
   END_RUNG
   RUNG wire#w1
      Contact( #Mx_ET51 )
   END_RUNG wire#w3
   RUNG wire#w1
      Contact( #Mx_ET60 )
      wire#w4
      Coil( #EstadoVI.Etapas_Descarga_S4 )
   END_RUNG
   RUNG wire#w1
      Contact( #Mx_ET61 )
   END_RUNG wire#w4
   RUNG wire#w1
      Contact( #Mx_ET70 )
      wire#w5
      Coil( #EstadoVI.Etapas_Descarga_S3 )
   END_RUNG
   RUNG wire#w1
      Contact( #Mx_ET71 )
   END_RUNG wire#w5
   // the same network as SCL:
   #EstadoVI.Etapas_Reset := "ON" AND #Mx_ET00;
   #EstadoVI.Etapa_Vacia := "ON" AND #Mx_ET01;
   #EstadoVI.Etapa_Cargada := "ON" AND #Mx_ET02;
   #EstadoVI.Etapas_Carga_E1 := "ON" AND (#Mx_ET10 OR #Mx_ET11);
   #EstadoVI.Etapas_Descarga_S2 := "ON" AND (#Mx_ET50 OR #Mx_ET51);
   #EstadoVI.Etapas_Descarga_S4 := "ON" AND (#Mx_ET60 OR #Mx_ET61);
   #EstadoVI.Etapas_Descarga_S3 := "ON" AND (#Mx_ET70 OR #Mx_ET71);
END_REGION

REGION Network 36: ENTRADAS DE LA MESA
   RUNG wire#powerrail
      Contact( TRUE )
      wire#w1
      Contact( #Error_Tx )
      Coil( #EstadoVI.En_Termico1 )
   END_RUNG
   RUNG wire#w1
      Contact( #pHsMx )
      Coil( #EstadoVI.En_PHS_1 )
   END_RUNG
   RUNG wire#w1
      Contact( #TP_Up )
      Coil( #EstadoVI.En_Tope1_UP )
   END_RUNG
   RUNG wire#w1
      Contact( #TP_Down )
      Coil( #EstadoVI.En_Tope1_DOWN )
   END_RUNG
   // the same network as SCL:
   #EstadoVI.En_Termico1 := TRUE AND #Error_Tx;
   #EstadoVI.En_PHS_1 := TRUE AND #pHsMx;
   #EstadoVI.En_Tope1_UP := TRUE AND #TP_Up;
   #EstadoVI.En_Tope1_DOWN := TRUE AND #TP_Down;
END_REGION

REGION Network 37: SALIDAS DE LA MESA
   RUNG wire#powerrail
      Contact( TRUE )
      wire#w1
      Contact( "DB1_SalidasExterioresDeMesa".Mesa[#Mesa].Avanzar_E1E3 )
      Contact( #Avance_Tx )
      Coil( #EstadoVI.Sa_Rod_Avance )
   END_RUNG
   RUNG wire#w1
      Contact( "DB1_SalidasExterioresDeMesa".Mesa[#Mesa].Subir_TP_E1E3 )
      Coil( #EstadoVI.Sa_Tope1_Sub )
   END_RUNG
   RUNG wire#w1
      Contact( "DB1_SalidasExterioresDeMesa".Mesa[#Mesa].Bajar_TP_E1E3 )
      Coil( #EstadoVI.Sa_Tope1_Baj )
   END_RUNG
   // the same network as SCL:
   #EstadoVI.Sa_Rod_Avance := TRUE AND "DB1_SalidasExterioresDeMesa".Mesa[#Mesa].Avanzar_E1E3 AND #Avance_Tx;
   #EstadoVI.Sa_Tope1_Sub := TRUE AND "DB1_SalidasExterioresDeMesa".Mesa[#Mesa].Subir_TP_E1E3;
   #EstadoVI.Sa_Tope1_Baj := TRUE AND "DB1_SalidasExterioresDeMesa".Mesa[#Mesa].Bajar_TP_E1E3;
END_REGION

REGION Network 38: FINALIZAR - Guardar las Variables de Trabajo de la Mesa
   RUNG wire#powerrail
      Move(in := #EstadoVI, out1 => "DB900_Estado_Mesas".EstadoVI[#Mesa])
   END_RUNG
   // the same network as SCL:
   "DB900_Estado_Mesas".EstadoVI[#Mesa] := #EstadoVI;
END_REGION
END_FUNCTION_BLOCK
